FUNCTION_BLOCK InRange (* Basic Function Block Type *)
  (* Standard: 61499-2 *)
  (* Version 0.0, 9/14/2008, Horst Mayer, nxtControl GmbH, Template *)
  PACKAGE Main;
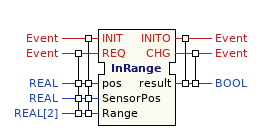
  EVENT_INPUT
    INIT WITH pos, SensorPos, Range; (* Initialization Request *)
    REQ WITH pos, SensorPos, Range; (* Normal Execution Request *)
  END_EVENT
  EVENT_OUTPUT
    INITO WITH result; (* Initialization Confirm *)
    CHG WITH result; (* Execution Confirmation *)
  END_EVENT
  VAR_INPUT
    pos : REAL;
    SensorPos : REAL;
    Range : ARRAY [0..1] OF REAL;
  END_VAR
  VAR_OUTPUT
    result : BOOL;
  END_VAR
  VAR
    presult : BOOL;
  END_VAR
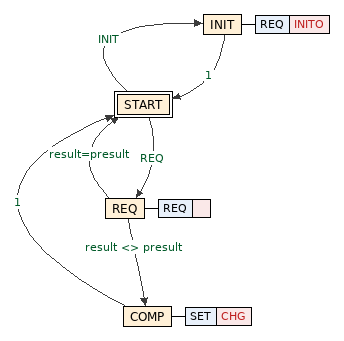
  EC_STATES
    START; (* Initial State *)
    INIT : REQ -> INITO; (* Initialization *)
    REQ : REQ; (* Normal execution *)
    COMP : SET -> CHG;
  END_STATES
  EC_TRANSITIONS
    START TO INIT := INIT;
    INIT TO START := 1;
    START TO REQ := REQ;
    REQ TO COMP := result <> presult;
    COMP TO START := 1;
    REQ TO START := result=presult;
  END_TRANSITIONS
  ALGORITHM SET IN ST: (* Initialization algorithm *)
 presult := result;
;
  END_ALGORITHM
  ALGORITHM REQ IN ST: (* Normally executed algorithm *)
IF (pos >= Range[0] + SensorPos) AND (pos <= Range[1] + SensorPos) THEN
 result := TRUE;
ELSE
 result := FALSE;
END_IF;
  END_ALGORITHM
END_FUNCTION_BLOCK
